Yaskawa INFORM job: SCANNING2.JBI

/JOB
//NAME SCANNING2
//POS
///NPOS 0,0,0,0,0,0
//INST
///DATE 2023/01/29 16:25
///ATTR SC,RW
///GROUP1 RB1,ST1
NOP
END
